(* CODESYS project cl_greenhouseobjectslibrary.library
   Author: Massimo Lucano
   Placeholder: CL_GreenhouseObjects
   Title: CL_GreenhouseObjectsLibrary
   Version: 1.3.3
   Description: library containing all class related to Greenhouse harware objects
   Company: CleanGreensSA

Project tree, tasks and I/O mapping:
  libraries: DefectManager_class, * (CleanGreensSA); Tc2_Standard, * (Beckhoff Automation GmbH); Tc2_System, * (Beckhoff Automation GmbH); Tc3_Module, * (Beckhoff Automation GmbH)
  DUTs/
    data type E_ModeMachine
    data type E_SeqLoader
    data type E_StateMachine
    data type ST_FrqCnvrCtrl_HWQ
    data type ST_StackLight_HWQ
  GVLs/
    global variables C
  POUs/
    ClassesObjectsHW/
      Classes_greeenhouse_20240729/
        function block CL_ButtonBlink [ST]: BlinkOff, BlinkOn, bPressed, Init, LightOff, LightOn
        function block CL_DoubleStopper [ST]: bDesactiveError, bInError, bIsBusyDown, bIsBusyUp, bIsDone, bIsDown, bIsNotDown, bIsUp, Init, InitDefect, ReqDown, ReqUp
        function block CL_Lift_old [ST]: bDesactiveError, bInError, bIsBusyDown, bIsBusyUp, bIsDone, bIsDown, bIsNotDown, bIsUp, Init, ReqDown, ReqUp
        function block CL_LiftStopper [ST]: bDesactiveError, bInError, bIsBusyDown, bIsBusyUp, bIsDone, bIsDown, bIsNotDown, bIsUp, DefectUpdate, Init, InitDefect, ReqDown, ReqUp, Run
        function block CL_LoaderOld [ST]: bInError, bIsBusy, bIsDone, bIsLoad, Init, InitDefect, ReqExtend, ReqLoad, ReqRetract, ReqStop
        function EMPTYSTR2 [ST]
        function FC_TransferPointer [ST]
      function block CL_Ancestor [ST]: Case01Hysto, Case02Hysto, Case03Hysto
      function block CL_Button [ST]: bPressed, Init, LightOff, LightOn
      function block CL_ButtonSafe [ST]: BtnPressed, BtnReleased, Init, LightOff, LightOn
      function block CL_Debug [ST]: Case01Histo, Case02Histo, Case03Histo
      function block CL_FrequencyConverter [ST]: bIsReady, bIsStopped, bSpeedReached, FB_init, Init, ReqMoveBW, ReqMoveFW, ReqReset, ReqStop
      function block CL_GreenhouseSystem [ST]: nModeMachine, nStateMachine, ReqModeMachine
      function block CL_LiftValvesBistableClosed [ST]: bIsBusyDown, bIsBusyUp, bIsDone, bIsDown, bIsUp, Init, ReqDown, ReqUp
      function block CL_SensorFilter [ST]: bStatus, DoNotTouch, FB_init, Init
      function block CL_StackLight [ST]: Init
      function block CL_WaitTimer [ST]: End, Start
      function block CL_WorkbenchRedLight [ST]: BlinkingRed, Init, RedOff, RedOn, Run
      function block CL_WorkbenchSensor [ST]: Init, isModule
      function block CL_WorkbenchStackLight [ST]: Blink, BlinkingOrange, Green, Init, Orange, redOnly, startBlinkingError, stopBlinkingError
  VISUs/
*)

// DUTs/E_ModeMachine
{attribute 'qualified_only'}
{attribute 'strict'}
TYPE E_ModeMachine :
(
  Automatic := 0,
  Manual,
  Startup,
  Setup,
  Maintenance,
  Disabled
);
END_TYPE

// DUTs/E_SeqLoader
{attribute 'qualified_only'}
{attribute 'strict'}
TYPE E_SeqLoader :
(
  cIdle           := 0,
  cStartExtend       ,
  cMovingExtend      ,
  cTargetReached      ,
  cStartRetract      ,
  cMovingRetract     ,
  cEndMovement        ,
  cError
);
END_TYPE

// DUTs/E_StateMachine
{attribute 'qualified_only'}
{attribute 'strict'}
TYPE E_StateMachine :
(
  cIdle := 0,
  cStarting,
  cExecute,
  cStopping,
  cStopped,
  cAborting,
  cAborted,
  cClearing,
  cResetting,
  cInitialization := 255        
);
END_TYPE

// DUTs/ST_FrqCnvrCtrl_HWQ
TYPE ST_FrqCnvrCtrl_HWQ :
STRUCT
  bMoveFW_gq     : BOOL;
  bMoveBW_gq     : BOOL;
  bHighSpeed_gq  : BOOL;
  bReset_gq      : BOOL;
END_STRUCT
END_TYPE

// DUTs/ST_StackLight_HWQ
TYPE ST_StackLight_HWQ :
STRUCT
  bBlue     : BOOL;
  bGreen    : BOOL;
  bOrange   : BOOL;
  bRed      : BOOL;
  bBuzzer   : BOOL;
END_STRUCT
END_TYPE

// GVLs/C
{attribute 'qualified_only'}
VAR_GLOBAL CONSTANT 
	//debug
	uiHistoStep_C								        : INT := 50;
	
	//LiftWorkbench Stacklight
	tLWBBlinkHalfPeriod_C               : TIME :=  T#350MS; // Used for every blinking stacklight
	
	//Lift constant
	//tLift_C													    : TIME := T#3S;

  //Lift error constant
	tLiftDown_C 											  : TIME := T#10S;
	tLiftUp_C  												  : TIME := T#10S;

  //Stopper error constant
	tStopperDown_C 											: TIME := T#5S;
	tStopperUp_C  											: TIME := T#5S;

  //Loader Constant
  tLoaderExtand_C                     : TIME := T#20S;
  tLoaderRetract_C                    : TIME := T#15S;

  //debug
	uiHistoryStep_C										  : INT := 50;
END_VAR

// POUs/ClassesObjectsHW/Classes_greeenhouse_20240729/CL_ButtonBlink
FUNCTION_BLOCK PUBLIC CL_ButtonBlink  EXTENDS R_trig
VAR
	bBtnSens_P 		: POINTER TO BOOL;
	bBtnLight_P 	: POINTER TO BOOL;
	bInit 				: BOOL := FALSE;
	bLight			 	: BOOL := FALSE;
	bBlink				: BOOL := FALSE;
  fbBlink     	: TON := (PT := T#0.5S);
	fbBlink2     	: TON := (PT := T#1.0S);
END_VAR

IF bInit THEN 
	SUPER^(CLK := bBtnSens_P^);
	fbBlink2(in := NOT fbBlink2.Q);
	fbBlink(in :=  fbBlink2.IN);
	
	IF bBlink THEN
		bBtnLight_P^:= fbBlink.Q;
	ELSE
		bBtnLight_P^:= bLight;
	END_IF

END_IF

METHOD PUBLIC BlinkOff
VAR_INPUT
END_VAR
IF bInit THEN 
	bBlink := FALSE;
	bLight := FALSE;
END_IF
END_METHOD

METHOD PUBLIC BlinkOn
VAR_INPUT
END_VAR
IF bInit THEN 
	bBlink := TRUE;
	bLight := FALSE;
END_IF
END_METHOD

PROPERTY PUBLIC bPressed : BOOL
GET
IF bInit THEN
	bPressed := SUPER^.Q;
	{IF defined (debug)}
	bPressed := bBtnSens_P^;
	{END_IF}
ELSE
	bPressed := false;
END_IF
END_GET
END_PROPERTY

METHOD PUBLIC Init : BOOL
VAR_INPUT
	bBtnSensPtrIn_P   : POINTER TO BOOL;
	bBtnLightPtrIn_P  : POINTER TO BOOL;
END_VAR
Init := FALSE;
IF NOT bInit THEN
	Init := bInit := bBtnSensPtrIn_P <> 0 AND bBtnLightPtrIn_P <> 0;
	bBtnSens_P := bBtnSensPtrIn_P;
	bBtnLight_P := bBtnLightPtrIn_P;
	bLight := FALSE;
	bBlink := FALSE;
END_IF
END_METHOD

METHOD PUBLIC LightOff
IF bInit THEN 
	bLight := FALSE;
	bBlink := FALSE; 
END_IF
END_METHOD

METHOD PUBLIC LightOn
IF bInit THEN 
	bLight := TRUE;
	bBlink := FALSE;
END_IF
END_METHOD

END_FUNCTION_BLOCK

// POUs/ClassesObjectsHW/Classes_greeenhouse_20240729/CL_DoubleStopper
(*
ExtractorStopper normally UP
PerpendStopper normally DOWN
controlled together by ExtractorDownPerpendUpStoppersVlv
ExtractorStopperDown and PerpendStopperDown
*)

(*
RFIDStopper normally UP
HandoverStopper normally DOWN
controlled together by RFIDDownHandoverUpStoppersVlv
RFIDStopperDown
*)

FUNCTION_BLOCK CL_DoubleStopper
VAR
//Defect
  objTimeOutStopperUp  : CL_Defect; (*	Not used, so no way to check if the object is working or not	*)
  objTimeOutStopperDown: CL_Defect;

//Error Var
	bErrorUp          : BOOL;
	bErrorDown        : BOOL;
  
//Seq management
	nstpMain          : INT := 0;
  nHistoryStm_AR    : ARRAY[0..C.uiHistoryStep_C] OF INT;
  nLastStm          : INT := -1;

//Index	
  i                 : INT;

//Other var 
  bInit             : BOOL;
  
//FBs
	fbTimerStopperUp     : TON ;
	fbErrorStopperDown   : TON := (PT:= C.tStopperDown_C);
	fbErrorStopperUp     : TON := (PT:= C.tStopperUp_C);
	
//Methods Request
	bRequUp           : BOOL;
	bRequDown         : BOOL;
  
// INTERNAL VAR 		
	_bSensorStp1Down					: BOOL;
  _bSensorStp1Down_P       	: POINTER TO BOOL;
  _bSensorStp2Down_P       	: POINTER TO BOOL;//the secondary stopper could have a down sensor
  _bValveUp_P          			: POINTER TO BOOL;
	
  _objGHSystem_P  : POINTER TO CL_GreenhouseSystem;
  _bIsBusy             : BOOL;
  _bIsBusyUP           : BOOL;
  _bIsBusyDown         : BOOL;
	_bIsDone             : BOOL;
  _bDesactiveError     : BOOL;
  _nLineNumber_P       : POINTER TO INT;
END_VAR

VAR CONSTANT
	nIdle_C             : INT := 0;
	WaitUP_C            : INT := 1;
	nWaitDown_C         : INT := 2;
	nLiftError_C        : INT := 3;
END_VAR

IF NOT bInit THEN
  RETURN;
END_IF

_bSensorStp1Down := _bSensorStp1Down_P^;

fbTimerStopperUp(IN:= NOT _bSensorStp1Down AND _bValveUp_P^);//sensor is false and valve is power on -> trigger timer IN from false to true rising edge

(*IF NOT _bDesactiveError THEN
	IF _objGHSystem_P^.nModeMachine <> E_ModeMachine.Manual THEN// desactive Error in manual mode
		fbErrorStopperUp(IN:= _bSensorStp1Down AND _bValveUp_P^);//stopper should go down -> if after the selected time Q is true --> stopper error remains UP
		fbErrorStopperDown(IN:= NOT _bSensorStp1Down AND NOT _bValveUp_P^);//stopper should go up -> if after the selected time Q is true --> stopper error remains DOWN
	END_IF
	
//	bErrorUp := fbErrorStopperUp.Q;
//	bErrorDown := fbErrorStopperDown.Q;
	objTimeOutStopperUp();
//	objTimeOutStopperUp.SetState(fbErrorStopperUp.Q);
	objTimeOutStopperDown();
//	objTimeOutStopperDown.SetState(fbErrorStopperDown.Q);
	
	IF bErrorUp OR bErrorDown THEN 
		bRequUP := bRequDown := FALSE;//cancel method request
		_bIsDone := FALSE;
		_bIsBusy := FALSE;
		_bIsBusyDown := FALSE;
		_bIsBusyUP := FALSE;
		nstpMain := nLiftError_C;
	END_IF
END_IF*)


CASE nstpMain OF
  // -------------------------------------------------
  nIdle_C:
    IF bRequUp THEN
      bRequUP := FALSE;
      nstpMain := WaitUP_C;
    ELSIF bRequDown THEN
      bRequDown := FALSE;
      nstpMain := nWaitDown_C;
    END_IF
  
  // -------------------------------------------------
  WaitUP_C:
    //lift is going up; no sensor available -> return true when calibration time elapsed
    _bValveUp_P^ := TRUE; //can power on electro-valve
    IF fbTimerStopperUp.Q  THEN
      //if after the calibrated time the sensor is true -> error lift is still down; error detected with the timer
      nstpMain := nIdle_C;
      _bIsDone := TRUE;
      _bIsBusy := FALSE;
      _bIsBusyUp := FALSE;
    END_IF
  
  // -------------------------------------------------
  nWaitDown_C:
    IF _bSensorStp1Down  THEN //lift is down -> sensor is true
      nstpMain := nIdle_C;
      _bIsDone := TRUE;
      _bIsBusy := FALSE;
      _bIsBusyDown := FALSE;
    ELSE
     _bValveUp_P^ := FALSE; //sensor is false -> can power off electro-valve
    END_IF
    
  // -------------------------------------------------
  nLiftError_C:
    //error handling lift error
    IF NOT bErrorUp AND  NOT bErrorDown THEN
      nstpMain := nIdle_C;
    END_IF
END_CASE

  
//Historization of STM
IF nLastStm <> nstpMain THEN
  nLastStm := nstpMain;
  FOR i := C.uiHistoryStep_C TO 1 BY -1 DO
    nHistoryStm_AR[i] := nHistoryStm_AR[i-1];
  END_FOR
  nHistoryStm_AR[0] := nstpMain;
END_IF

PROPERTY bDesactiveError : bool
GET
bDesactiveError := _bDesactiveError;
END_GET
SET
_bDesactiveError := bDesactiveError;
END_SET
END_PROPERTY

PROPERTY bInError : bool
GET
bInError := fbErrorStopperUp.Q OR fbErrorStopperDown.Q;
END_GET
END_PROPERTY

PROPERTY PUBLIC bIsBusyDown : bool
GET
bIsBusyDown := _bIsBusyDown;
END_GET
END_PROPERTY

PROPERTY PUBLIC bIsBusyUp : bool
GET
bIsBusyUp := _bIsBusyUp;
END_GET
END_PROPERTY

PROPERTY PUBLIC bIsDone : bool
GET
bIsDone := _bIsDone;
END_GET
END_PROPERTY

PROPERTY PUBLIC bIsDown : BOOL
GET
bIsDown := _bSensorStp1Down AND NOT _bValveUp_P^;//lift is in down position -> sensor is true and valve is power off  isIN
END_GET
END_PROPERTY

PROPERTY PUBLIC bIsNotDown : BOOL
GET
bIsNotDown := NOT bIsDown;//lift is not in down position -> sensor is true and valve is power off
END_GET
END_PROPERTY

PROPERTY PUBLIC bIsUp : bool
GET
bIsUp := fbTimerStopperUp.Q ;//elapsed time to assert that the stopper is in up position
{IF defined (debug)}
bIsUp := TRUE ;
{END_IF}
END_GET
END_PROPERTY

METHOD Init : BOOL
VAR_INPUT
  //Obj
  GHSystem_P 	: POINTER TO CL_GreenhouseSystem;
  
  //IO
  bSensorStp1Down_P	: POINTER TO BOOL;
  bSensorStp2Down_P	: POINTER TO BOOL;
  bValveStp1Up_P		: POINTER TO BOOL;

  //Var
	tStp1Up						: TIME;
	
	// Location number
	usiNbLocatStopper			: USINT;
END_VAR

// Class ID: 020
//Init Obj
_objGHSystem_P  := GHSystem_P ;

//Init IO
_bSensorStp1Down_P  := bSensorStp1Down_P;
_bSensorStp2Down_P  := bSensorStp2Down_P;//if set to NULL then no secondary sensor available
_bValveUp_P := bValveStp1Up_P;

//Init Var
Init := FALSE;
//Check Init
IF bSensorStp1Down_P <> 0 AND _bValveUp_P <> 0 AND _objGHSystem_P <> 0 THEN
  //Defect
//  ObjTimeOutStopperUp.Register(gvl.objDefectManager,CidCL.sClassID_DoubleStopper_C[usiNbLocatStopper],CidErr.sErrorIDs_DoubleStopper_C[1]);
//  ObjTimeOutStopperDown.Register(gvl.objDefectManager,CidCL.sClassID_DoubleStopper_C[usiNbLocatStopper],CidErr.sErrorIDs_DoubleStopper_C[2]);
  InitDefect(iNumInst := usiNbLocatStopper); // Conversion from short unsigned to signed integer always possible, so OK.
	
  Init := bInit := TRUE;
	fbTimerStopperUp.PT := tStp1Up;	// Maybe to move inside the InitDefect method
END_IF
END_METHOD

METHOD InitDefect : BOOL
VAR_INPUT
	iNumInst	:	INT;
END_VAR
END_METHOD

METHOD PUBLIC ReqDown : BOOL
ReqDown := FALSE;

IF NOT bInError THEN
  ReqDown := TRUE;
  bRequDown := TRUE;
  _bIsBusy := TRUE;
  _bIsBusyDown := TRUE;
END_IF

_bIsDone := FALSE;
END_METHOD

METHOD ReqUp : BOOL
ReqUp := FALSE;

IF NOT bInError THEN
  ReqUp := TRUE;
  bRequUp := TRUE;
  _bIsBusy := TRUE;
  _bIsBusyUp := TRUE;
END_IF

_bIsDone := FALSE;
END_METHOD

END_FUNCTION_BLOCK

// POUs/ClassesObjectsHW/CL_GreenhouseSystem
FUNCTION_BLOCK CL_GreenhouseSystem extends CL_Ancestor
VAR_INPUT
END_VAR
VAR_OUTPUT
END_VAR
VAR
  nLastStateMachine         : E_StateMachine;
  nHistoStateMachine_AR     : ARRAY[0..100]OF E_StateMachine;
  //z                         : UINT;
  
  //INTERNAL VAR
  _nRequestModeMachine      : E_ModeMachine := E_ModeMachine.Automatic;
  _nModeMachine             : E_ModeMachine := E_ModeMachine.Automatic;
  _nStateMachine            : E_StateMachine := E_StateMachine.cIdle;
END_VAR

//State machine histroy
IF nLastStateMachine <> nStateMachine THEN
  nLastStateMachine := nStateMachine;  
  Case01Hysto(nStateMachine);
END_IF

//Manage Mode machine
IF _nRequestModeMachine <> nModeMachine AND _nStateMachine = E_StateMachine.cStopped THEN
	_nModeMachine := _nRequestModeMachine;
END_IF

PROPERTY nModeMachine : E_ModeMachine
GET
nModeMachine := _nModeMachine;
END_GET
SET
_nModeMachine := nModeMachine;
END_SET
END_PROPERTY

PROPERTY nStateMachine : E_StateMachine
GET
nStateMachine := _nStateMachine;
END_GET
SET
_nStateMachine := nStateMachine;
END_SET
END_PROPERTY

METHOD ReqModeMachine : BOOL
VAR_INPUT
  nModeMachine   :E_ModeMachine;
END_VAR
_nRequestModeMachine := nModeMachine;
END_METHOD

END_FUNCTION_BLOCK

// POUs/ClassesObjectsHW/CL_Ancestor
FUNCTION_BLOCK CL_Ancestor
VAR
	i01                         : INT;
  nHistoryStep_AR01           : ARRAY[0..C.uiHistoStep_C] OF DINT;
  nLastStep01                 : DINT := -1;
  
  i02                         : INT;
  nHistoryStep_AR02           : ARRAY[0..C.uiHistoStep_C] OF DINT;
  nLastStep02                 : DINT := -1;
  
  i03                         : INT;
  nHistoryStep_AR03           : ARRAY[0..C.uiHistoStep_C] OF DINT;
  nLastStep03                 : DINT := -1;
END_VAR

METHOD Case01Hysto : BOOL
VAR_INPUT
	nStep : DINT;
END_VAR
IF nStep <> nLastStep01 THEN
  nLastStep01 := nStep;
  FOR i01:= C.uiHistoStep_C TO 1 BY -1 DO
    nHistoryStep_AR01[i01] := nHistoryStep_AR01[i01-1];
  END_FOR
  nHistoryStep_AR01[0] := nStep;
END_IF
END_METHOD

METHOD Case02Hysto : BOOL
VAR_INPUT
	nStep : DINT;
END_VAR
IF nStep <> nLastStep02 THEN
  nLastStep02 := nStep;
  FOR i02:= C.uiHistoStep_C TO 1 BY -1 DO
    nHistoryStep_AR02[i02] := nHistoryStep_AR01[i02-1];
  END_FOR
  nHistoryStep_AR02[0] := nStep;
END_IF
END_METHOD

METHOD Case03Hysto : BOOL
VAR_INPUT
	nStep : DINT;
END_VAR
IF nStep <> nLastStep03 THEN
  nLastStep03 := nStep;
  FOR i03:= C.uiHistoStep_C TO 1 BY -1 DO
    nHistoryStep_AR03[i03] := nHistoryStep_AR01[i03-1];
  END_FOR
  nHistoryStep_AR03[0] := nStep;
END_IF
END_METHOD

END_FUNCTION_BLOCK

// POUs/ClassesObjectsHW/Classes_greeenhouse_20240729/CL_Lift_old
FUNCTION_BLOCK CL_Lift_old
VAR
//Defect
  objTimeOutLiftUp  : CL_Defect;
  objTimeOutLiftDown: CL_Defect;

//Error Var
	bErrorUp          : BOOL;
	bErrorDown        : BOOL;
  
//Seq management
	nstpMain          : INT := 0;
  nHistoryStm_AR    : ARRAY[0..C.uiHistoryStep_C] OF INT;
  nLastStm          : INT := -1;

//Index	
	i                	: UINT;
  hi                : INT;

//Other var 
  bInit             : BOOL;
  
//FBs
	fbTimerLiftUp     : TON ;
	fbErrorLiftDown   : TON := (PT:= C.tLiftDown_C);
	fbErrorLiftUp     : TON := (PT:= C.tLiftUp_C);
	
//Methods Request
	bRequUp           : BOOL;
	bRequDown         : BOOL;
  
// INTERNAL VAR 
  _bSensorDown_P       : POINTER TO BOOL;
  _bValveUp_P          : POINTER TO BOOL;
  _objGHSystem_P  : POINTER TO CL_GreenhouseSystem;
  _bIsBusy             : BOOL;
  _bIsBusyUP           : BOOL;
  _bIsBusyDown         : BOOL;
	_bIsDone             : BOOL;
  _bDesactiveError     : BOOL;
  _nLineNumber_P       : POINTER TO INT;
END_VAR

VAR CONSTANT
	nIdle_C             : INT := 0;
	WaitUP_C            : INT := 1;
	nWaitDown_C         : INT := 2;
	nLiftError_C        : INT := 3;
END_VAR

IF NOT bInit THEN
  RETURN;
END_IF

fbTimerLiftUp(IN:= NOT _bSensorDown_P^ AND _bValveUp_P^);//sensor is false and valve is power on -> trigger timer IN from false to true rising edge

IF NOT _bDesactiveError THEN
	IF _objGHSystem_P^.nModeMachine <> E_ModeMachine.Manual THEN// desactive Error in manual mode
		fbErrorLiftUp(IN:= _bSensorDown_P^ AND _bValveUp_P^);//lift should going down -> if after the selected time Q is true --> lift error remains UP
		fbErrorLiftDown(IN:= NOT _bSensorDown_P^ AND NOT _bValveUp_P^);//lift should going up -> if after the selected time Q is true --> lift error remains DOWN
	END_IF
	
	bErrorUp := fbErrorLiftUp.Q;
	bErrorDown := fbErrorLiftDown.Q;
	ObjTimeOutLiftUp();
	ObjTimeOutLiftUp.Set(fbErrorLiftUp.Q);
	ObjTimeOutLiftDown();
	ObjTimeOutLiftDown.Set(fbErrorLiftDown.Q);
	
	IF bErrorUp OR bErrorDown THEN 
		bRequUP := bRequDown := FALSE;//cancel method request
		_bIsDone := FALSE;
		_bIsBusy := FALSE;
		_bIsBusyDown := FALSE;
		_bIsBusyUP := FALSE;
		nstpMain := nLiftError_C;
	END_IF
end_if


CASE nstpMain OF
  // -------------------------------------------------
  nIdle_C:
    IF bRequUp THEN
      bRequUP := FALSE;
      nstpMain := WaitUP_C;
    ELSIF bRequDown THEN
      bRequDown := FALSE;
      nstpMain := nWaitDown_C;
    END_IF
  
  // -------------------------------------------------
  WaitUP_C:
    //lift is going up; no sensor available -> return true when calibration time elapsed
    _bValveUp_P^ := TRUE; //can power on electro-valve
    IF fbTimerLiftUp.Q  THEN
      //if after the calibrated time the sensor is true -> error lift is still down; error detected with the timer
      nstpMain := nIdle_C;
      _bIsDone := TRUE;
      _bIsBusy := FALSE;
      _bIsBusyUp := FALSE;
    END_IF
  
  // -------------------------------------------------
  nWaitDown_C:
    IF _bSensorDown_P^  THEN //lift is down -> sensor is true
      nstpMain := nIdle_C;
      _bIsDone := TRUE;
      _bIsBusy := FALSE;
      _bIsBusyDown := FALSE;
    ELSE
     _bValveUp_P^ := FALSE; //sensor is false -> can power off electro-valve
    END_IF
    
  // -------------------------------------------------
  nLiftError_C:
    //error handling lift error
    IF NOT bErrorUp AND  NOT bErrorDown THEN
      nstpMain := nIdle_C;
    END_IF
END_CASE

  
//Historization of STM
IF nLastStm <> nstpMain THEN
  nLastStm := nstpMain;
  FOR hi := C.uiHistoryStep_C TO 1 BY -1 DO
    nHistoryStm_AR[hi] := nHistoryStm_AR[hi-1];
  END_FOR
  nHistoryStm_AR[0] := nstpMain;
END_IF

PROPERTY bDesactiveError : bool
GET
bDesactiveError := _bDesactiveError;
END_GET
SET
_bDesactiveError := bDesactiveError;
END_SET
END_PROPERTY

PROPERTY bInError : bool
GET
bInError := fbErrorLiftUp.Q or fbErrorLiftDown.Q;
END_GET
END_PROPERTY

PROPERTY PUBLIC bIsBusyDown : bool
GET
bIsBusyDown := _bIsBusyDown;
END_GET
END_PROPERTY

PROPERTY PUBLIC bIsBusyUp : bool
GET
bIsBusyUp := _bIsBusyUp;
END_GET
END_PROPERTY

PROPERTY PUBLIC bIsDone : bool
GET
bIsDone := _bIsDone;
END_GET
END_PROPERTY

PROPERTY PUBLIC bIsDown : BOOL
GET
bIsDown := _bSensorDown_P^ AND NOT _bValveUp_P^;//lift is in down position -> sensor is true and valve is power off  isIN
END_GET
END_PROPERTY

PROPERTY PUBLIC bIsNotDown : BOOL
GET
bIsNotDown := NOT bIsDown;//lift is not in down position -> sensor is true and valve is power off
END_GET
END_PROPERTY

PROPERTY PUBLIC bIsUp : bool
GET
bIsUp := fbTimerLiftUp.Q ;//elapsed time to assert that the lift is in up position
{IF defined (debug)}
//bIsUp := TRUE ;
{END_IF}
END_GET
END_PROPERTY

METHOD Init : BOOL
VAR_INPUT
  //Obj
  objGHSystem_P : POINTER TO CL_GreenhouseSystem;
  
  //IO
  bSensorDown_P	: POINTER TO BOOL;
  bValveUp_P		: POINTER TO BOOL;
  //Var
	tLiftUp				: TIME;
  nLineNumber_P : POINTER TO INT;
END_VAR
//Init Obj
_objGHSystem_P  := objGHSystem_P;

//Init IO
_bSensorDown_P  := bSensorDown_P;
_bValveUp_P := bValveUp_P;

//Init Var
_nLineNumber_P := nLineNumber_P;

Init := FALSE;
//Check Init
IF _bSensorDown_P <> 0 AND _bValveUp_P <> 0 AND _objGHSystem_P <> 0 AND _nLineNumber_P <> 0 THEN
  //Defect
//  ObjTimeOutLiftUp.Register(gvl.objDefectManager,CidCL.sClassID_Lift_C[(_nLineNumber_P^)+C.usiNbLiftOutSpan_C],CidErr.sErrorIDs_Lift_C[1]);
//  ObjTimeOutLiftDown.Register(gvl.objDefectManager,CidCL.sClassID_Lift_C[(_nLineNumber_P^)+C.usiNbLiftOutSpan_C],CidErr.sErrorIDs_Lift_C[2]);
	
	// No InitDefect, since not intended to be used anymore (replaced by CL_Lift_new (which will be renamed CL_Lift in the end)).
//  ObjTimeOutLiftUp.Register(gvl.objDefectManager,CidCL.sClassID_Lift_C[(_nLineNumber_P^)+C.usiNbLiftOutSpan_C],CidErr.sLiftRiseTimeout);
//  ObjTimeOutLiftDown.Register(gvl.objDefectManager,CidCL.sClassID_Lift_C[(_nLineNumber_P^)+C.usiNbLiftOutSpan_C],CidErr.sLiftFallTimeout);
	// Reimplementation of the Defect, to avoid any overflow with the new error Ids for the Lifts
	ObjTimeOutLiftUp.Register(gvl.objDefectManager,CidCL.sClassID_Lift_C[_nLineNumber_P^],CidErr.sLiftRiseTimeout);
  ObjTimeOutLiftDown.Register(gvl.objDefectManager,CidCL.sClassID_Lift_C[_nLineNumber_P^],CidErr.sLiftFallTimeout);
	
  Init := bInit := TRUE;
	fbTimerLiftUp.PT := tLiftUp;
END_IF
END_METHOD

METHOD PUBLIC ReqDown : BOOL
ReqDown := FALSE;

IF NOT bInError THEN
  ReqDown := TRUE;
  bRequDown := TRUE;
  _bIsBusy := TRUE;
  _bIsBusyDown := TRUE;
END_IF

_bIsDone := FALSE;
END_METHOD

METHOD ReqUp : BOOL
ReqUp := FALSE;

IF NOT bInError THEN
  ReqUp := TRUE;
  bRequUp := TRUE;
  _bIsBusy := TRUE;
  _bIsBusyUp := TRUE;
END_IF

_bIsDone := FALSE;
END_METHOD

END_FUNCTION_BLOCK

// POUs/ClassesObjectsHW/Classes_greeenhouse_20240729/CL_LiftStopper
FUNCTION_BLOCK CL_LiftStopper
VAR
//Error Var
	bErrorUp          : BOOL;
	bErrorDown        : BOOL;
  
//Seq management
	nstpMain          : INT := 0;
  nHistoryStm_AR    : ARRAY[0..C.uiHistoryStep_C] OF INT;
  nLastStm          : INT := -1;

//Index	
	i                	: UINT;
  hi                : INT;

//Other var 
  bInit             : BOOL;
  
//FBs
	fbTimerLiftUp     : TON ;
	fbErrorLiftDown   : TON := (PT:= C.tLiftDown_C);
	fbErrorLiftUp     : TON := (PT:= C.tLiftUp_C);
	
//Methods Request
	bRequUp           : BOOL;
	bRequDown         : BOOL;
  
// INTERNAL VAR 
  _bSensorDown_P       : POINTER TO BOOL;
  _bValveUp_P          : POINTER TO BOOL;
  _objGHSystem_P  : POINTER TO CL_GreenhouseSystem;
  _bIsBusy             : BOOL;
  _bIsBusyUP           : BOOL;
  _bIsBusyDown         : BOOL;
	_bIsDone             : BOOL;
  _bDesactiveError     : BOOL;
  _nLineNumber_P       : POINTER TO INT;
	
	// Defect (common to all type of lift)
	objTimeOutAnyLiftUp  : CL_Defect;	// For every single valve, independent lift
  objTimeOutAnyLiftDown: CL_Defect;
END_VAR

VAR CONSTANT
	nIdle_C             : INT := 0;	// To replace by an enum!
	WaitUP_C            : INT := 1;
	nWaitDown_C         : INT := 2;
	nLiftError_C        : INT := 3;
END_VAR

THIS^.Run();

PROPERTY bDesactiveError : bool
GET
bDesactiveError := _bDesactiveError;
END_GET
SET
_bDesactiveError := bDesactiveError;
END_SET
END_PROPERTY

PROPERTY bInError : bool
GET
bInError := fbErrorLiftUp.Q or fbErrorLiftDown.Q;
END_GET
END_PROPERTY

PROPERTY PUBLIC bIsBusyDown : bool
GET
bIsBusyDown := _bIsBusyDown;
END_GET
END_PROPERTY

PROPERTY PUBLIC bIsBusyUp : bool
GET
bIsBusyUp := _bIsBusyUp;
END_GET
END_PROPERTY

PROPERTY PUBLIC bIsDone : bool
GET
bIsDone := _bIsDone;
END_GET
END_PROPERTY

PROPERTY PUBLIC bIsDown : BOOL
GET
bIsDown := _bSensorDown_P^ AND NOT _bValveUp_P^;//lift is in down position -> sensor is true and valve is power off  isIN
END_GET
END_PROPERTY

PROPERTY PUBLIC bIsNotDown : BOOL
GET
bIsNotDown := NOT bIsDown;//lift is not in down position -> sensor is true and valve is power off
END_GET
END_PROPERTY

PROPERTY PUBLIC bIsUp : bool
GET
bIsUp := fbTimerLiftUp.Q ;//elapsed time to assert that the lift is in up position
{IF defined (debug)}
//bIsUp := TRUE ;
{END_IF}
END_GET
END_PROPERTY

METHOD DefectUpdate : BOOL
END_METHOD

METHOD Init : BOOL
VAR_INPUT
  //Obj
  objGHSystem_P : POINTER TO CL_GreenhouseSystem;
  
  //IO
  bSensorDown_P	: POINTER TO BOOL;
  bValveUp_P		: POINTER TO BOOL;
  //Var
	tLiftUp				: TIME;
  nLineNumber_P : POINTER TO INT;
END_VAR
//Init Obj
_objGHSystem_P  := objGHSystem_P;

//Init IO
_bSensorDown_P  := bSensorDown_P;
_bValveUp_P := bValveUp_P;

//Init Var
_nLineNumber_P := nLineNumber_P;

Init := FALSE;
//Check Init
IF _bSensorDown_P <> 0 AND _bValveUp_P <> 0 AND _objGHSystem_P <> 0 AND _nLineNumber_P <> 0 THEN	// Not rightly written
	fbTimerLiftUp.PT := tLiftUp;	// To move inside the InitDefect ? No, but to replace if the same input in any case! Or keep it for sake of clarity.
  THIS^.InitDefect(iNumInst :=  nLineNumber_P^);	// Init to stabilise
	
	// To decide right now, but level to warning
  Init := bInit := TRUE;
END_IF
END_METHOD

METHOD InitDefect : BOOL
VAR_INPUT
	iNumInst	:	INT;
END_VAR
END_METHOD

METHOD PUBLIC ReqDown : BOOL
ReqDown := FALSE;

IF NOT bInError THEN
  ReqDown := TRUE;
  bRequDown := TRUE;
  _bIsBusy := TRUE;
  _bIsBusyDown := TRUE;
END_IF

_bIsDone := FALSE;
END_METHOD

METHOD ReqUp : BOOL
ReqUp := FALSE;

IF NOT bInError THEN
  ReqUp := TRUE;
  bRequUp := TRUE;
  _bIsBusy := TRUE;
  _bIsBusyUp := TRUE;
END_IF

_bIsDone := FALSE;
END_METHOD

METHOD Run : BOOL
VAR_INPUT
END_VAR
IF NOT bInit THEN
  RETURN;
END_IF

fbTimerLiftUp(IN:= NOT _bSensorDown_P^ AND _bValveUp_P^);//sensor is false and valve is power on -> trigger timer IN from false to true rising edge

IF NOT _bDesactiveError THEN
	IF _objGHSystem_P^.nModeMachine <> E_ModeMachine.Manual THEN// desactive Error in manual mode
		fbErrorLiftUp(IN:= _bSensorDown_P^ AND _bValveUp_P^);//lift should going down -> if after the selected time Q is true --> lift error remains UP
		fbErrorLiftDown(IN:= NOT _bSensorDown_P^ AND NOT _bValveUp_P^);//lift should going up -> if after the selected time Q is true --> lift error remains DOWN
	END_IF
	
	bErrorUp := fbErrorLiftUp.Q;
	bErrorDown := fbErrorLiftDown.Q;
	ObjTimeOutAnyLiftUp();
	ObjTimeOutAnyLiftUp.Set(fbErrorLiftUp.Q);
	ObjTimeOutAnyLiftDown();
	ObjTimeOutAnyLiftDown.Set(fbErrorLiftDown.Q);

	
	IF bErrorUp OR bErrorDown THEN 
		bRequUP := bRequDown := FALSE;//cancel method request
		_bIsDone := FALSE;
		_bIsBusy := FALSE;
		_bIsBusyDown := FALSE;
		_bIsBusyUP := FALSE;
		nstpMain := nLiftError_C;
	END_IF
end_if


CASE nstpMain OF
  // -------------------------------------------------
  nIdle_C:
    IF bRequUp THEN
      bRequUP := FALSE;
      nstpMain := WaitUP_C;
    ELSIF bRequDown THEN
      bRequDown := FALSE;
      nstpMain := nWaitDown_C;
    END_IF
  
  // -------------------------------------------------
  WaitUP_C:
    //lift is going up; no sensor available -> return true when calibration time elapsed
    _bValveUp_P^ := TRUE; //can power on electro-valve
    IF fbTimerLiftUp.Q  THEN
      //if after the calibrated time the sensor is true -> error lift is still down; error detected with the timer
      nstpMain := nIdle_C;
      _bIsDone := TRUE;
      _bIsBusy := FALSE;
      _bIsBusyUp := FALSE;
    END_IF
  
  // -------------------------------------------------
  nWaitDown_C:
    IF _bSensorDown_P^  THEN //lift is down -> sensor is true
      nstpMain := nIdle_C;
      _bIsDone := TRUE;
      _bIsBusy := FALSE;
      _bIsBusyDown := FALSE;
    ELSE
     _bValveUp_P^ := FALSE; //sensor is false -> can power off electro-valve
    END_IF
    
  // -------------------------------------------------
  nLiftError_C:
    //error handling lift error
    IF NOT bErrorUp AND  NOT bErrorDown THEN
      nstpMain := nIdle_C;
    END_IF
END_CASE

  
//Historization of STM
IF nLastStm <> nstpMain THEN
  nLastStm := nstpMain;
  FOR hi := C.uiHistoryStep_C TO 1 BY -1 DO
    nHistoryStm_AR[hi] := nHistoryStm_AR[hi-1];
  END_FOR
  nHistoryStm_AR[0] := nstpMain;
END_IF
END_METHOD

END_FUNCTION_BLOCK

// POUs/ClassesObjectsHW/Classes_greeenhouse_20240729/CL_LoaderOld
FUNCTION_BLOCK CL_LoaderOld
VAR
// Defect
  objTimeOutRetractDefect   :CL_Defect;
  objTimeOutExtandDefect    :CL_Defect;
  
// FBs
  fbTimeOutExtand           : TON :=(PT := c.tLoaderExtand_C);
  fbTimeOutRetract          : TON :=(PT := c.tLoaderRetract_C);
  fbTimeBeforeHighSpeed		  : TON := (PT := T#3S);
  fbTrigAbort               : R_TRIG;
  
// Request  
  bRequestLoad              : BOOL := FALSE;
  boRequestRetract          : BOOL := FALSE;
  boRequestExtend           : BOOL := FALSE;
  boOnlyExtend              : BOOL := FALSE;
  
// Seq management  
  nStep                     : INT := 0;
  nHistoryStep_AR           : ARRAY[0..C.uiHistoryStep_C] OF INT;
  nLastStep                 : INT := -1;
    
// Index  
  i                         : UINT;
	hi												: INT;

// Other var
  bInit                     : BOOL;
  
// INTERNAL VAR
  _bSensorIsExtend_P         : POINTER TO BOOL;
  _bSensorIsRetract_P        : POINTER TO BOOL;
  _bIsBusy                   : BOOL;
  _bIsDone                   : BOOL;  
  _bIsLoad                   : BOOL;
  _nLineNumber               : POINTER TO INT;
  
// INTERNAL OBJECT  
  _objPusher_P               : POINTER TO CL_FrequencyConverter;
  _objGHSystem_P     : POINTER TO CL_GreenhouseSystem;
END_VAR

IF NOT bInit THEN
  RETURN;
END_IF

//Call FBs
fbTimeOutExtand();
fbTimeOutRetract();
fbTimeBeforeHighSpeed(in :=nStep = E_SeqLoader.cMovingExtend);

//Defect
ObjTimeOutRetractDefect();
ObjTimeOutRetractDefect.Set(fbTimeOutRetract.Q);
ObjTimeOutExtandDefect();
ObjTimeOutExtandDefect.Set(fbTimeOutExtand.Q);

fbTrigAbort(CLK := _objGHSystem_P^.nStateMachine = E_StateMachine.cAborting);
IF fbTrigAbort.Q THEN
  nStep           := E_SeqLoader.cError;
  bRequestLoad     := FALSE;
  boRequestRetract := FALSE;
  boRequestExtend  := FALSE;
END_IF
IF _objGHSystem_P^.nStateMachine = E_StateMachine.cStopped THEN
  bRequestLoad     := FALSE;
  boRequestRetract := FALSE;
  boRequestExtend  := FALSE;
END_IF

//--------------------------------------------Sequence-----------------------------------------
CASE nStep OF
  // -------------------------------------------------
  E_SeqLoader.cIdle :
    IF boRequestExtend THEN
      boRequestExtend := FALSE;
      boOnlyExtend    := TRUE;
      nStep          := E_SeqLoader.cStartExtend;
     ELSIF boRequestRetract THEN
      boRequestRetract := FALSE;
      nStep          := E_SeqLoader.cStartRetract; 
     ELSIF bRequestLoad  THEN
      bRequestLoad := FALSE;
      nStep        := E_SeqLoader.cStartExtend;
		END_IF
    
  // -------------------------------------------------
  E_SeqLoader.cStartExtend :
    _objPusher_P^.ReqMoveBW(bHighSpeed:= FALSE);
    IF _bSensorIsExtend_P^  THEN
      nStep := E_SeqLoader.cTargetReached;
    ELSIF _objPusher_P^.bSpeedReached THEN       
      nStep := E_SeqLoader.cMovingExtend;
		END_IF
    
  // -------------------------------------------------
  E_SeqLoader.cMovingExtend :
  IF fbTimeBeforeHighSpeed.Q AND NOT _bSensorIsExtend_P^ THEN
	  _objPusher_P^.ReqMoveBW(bHighSpeed:= TRUE);
  END_IF
    IF fbTimeOutExtand.Q THEN
      nStep := E_SeqLoader.cError;
		END_IF
    IF _bSensorIsExtend_P^ THEN  
      _bIsLoad     := TRUE;
      nStep := E_SeqLoader.cTargetReached;
		END_IF
    
  // -------------------------------------------------
  E_SeqLoader.cTargetReached :
    _objPusher_P^.ReqStop();
    IF  _objPusher_P^.bIsStopped THEN
      IF boOnlyExtend THEN
        nStep := E_SeqLoader.cIdle;
        _bIsBusy     := FALSE;
        boOnlyExtend := FALSE;
      ELSE       
        nStep := E_SeqLoader.cStartRetract;
      END_IF
		END_IF
    
  // -------------------------------------------------
  E_SeqLoader.cStartRetract :
    _objPusher_P^.ReqMoveFW(bHighSpeed:= TRUE);
    IF _bSensorIsRetract_P^  THEN
      nStep := E_SeqLoader.cEndMovement;
    ELSIF _objPusher_P^.bSpeedReached THEN       
      nStep := E_SeqLoader.cMovingRetract;
		END_IF
    
  // -------------------------------------------------
  E_SeqLoader.cMovingRetract :
    IF fbTimeOutRetract.Q THEN
      nStep := E_SeqLoader.cError;
		END_IF
    IF _bSensorIsRetract_P^ THEN       
      nStep := E_SeqLoader.cEndMovement;
		END_IF
    
  // -------------------------------------------------
  E_SeqLoader.cEndMovement :
    _objPusher_P^.ReqStop();
    IF _objPusher_P^.bIsStopped THEN
      _bIsBusy  := FALSE;
      _bIsDone  := TRUE;
      nStep  := E_SeqLoader.cIdle;
		END_IF
    
  // -------------------------------------------------
  E_SeqLoader.cError :
    _bIsBusy  := FALSE;
    bRequestLoad := FALSE;
    _objPusher_P^.ReqStop();
    IF NOT _objPusher_P^.bIsReady AND _objPusher_P^.bIsStopped THEN
      _objPusher_P^.ReqReset();
    ELSE
      nStep  := E_SeqLoader.cIdle;
		END_IF
    
END_CASE


//Historization of the sequence
IF nLastStep <> nStep THEN
  nLastStep := nStep;
  FOR hi := C.uiHistoryStep_C TO 1 BY -1 DO
    nHistoryStep_AR[hi] := nHistoryStep_AR[hi-1];
  END_FOR
  nHistoryStep_AR[0] := nStep;
END_IF

PROPERTY bInError : bool
GET
bInError := nStep = E_SeqLoader.cError;
END_GET
END_PROPERTY

PROPERTY bIsBusy : BOOL
GET
bIsBusy := _bIsBusy;
END_GET
END_PROPERTY

PROPERTY bIsDone : BOOL
GET
bIsDone := _bIsDone;
END_GET
END_PROPERTY

PROPERTY bIsLoad : bool
GET
bIsLoad := _bIsLoad;
END_GET
END_PROPERTY

METHOD Init : BOOL
VAR_INPUT
  //Obj
  objPusher_P           : POINTER TO CL_FrequencyConverter;
  objGreenhouseSystem_P : POINTER TO CL_GreenhouseSystem;
  
  //IO
  bSensorIsExtend_P     : POINTER TO BOOL;
  bSensorIsRetract_P    : POINTER TO BOOL;
 
  //Var
  nLineNumber_P         : POINTER TO INT;
END_VAR

// Class ID: 040
//Init Obj
_objPusher_P := objPusher_P;
_objGHSystem_P := objGreenhouseSystem_P;

//Init IO
_bSensorIsExtend_P := bSensorIsExtend_P;
_bSensorIsRetract_P := bSensorIsRetract_P;

//Init Var
_nLineNumber := nLineNumber_P;

//Check Init
IF _objPusher_P <> 0 AND _bSensorIsExtend_P <> 0 AND _bSensorIsRetract_P <> 0 AND _objGHSystem_P <> 0 AND _nLineNumber <> 0 THEN
  //Defect
//  ObjTimeOutRetractDefect.Register(gvl.objDefectManager,CidCL.sClassID_Loader_C[(nLineNumber_P^)],CidErr.sErrorIDs_Loader_C[1]);
//  ObjTimeOutExtandDefect.Register(gvl.objDefectManager,CidCL.sClassID_Loader_C[(nLineNumber_P^)],CidErr.sErrorIDs_Loader_C[2]);
//  // CAUTION: not possible to indicate the line by this way
//  // => Future fix: use the location Infos in the database (maybe by using another stored procedure)
  InitDefect(iNumInst := nLineNumber_P^);
  bInit := TRUE;
END_IF
END_METHOD

METHOD InitDefect : BOOL
VAR_INPUT
	iNumInst	:	INT;
END_VAR
END_METHOD

METHOD ReqExtend : BOOL
VAR_INPUT
END_VAR
ReqExtend := FALSE;

IF _objPusher_P = 0 THEN
  RETURN;
END_IF

IF _objPusher_P^.bIsReady AND NOT bIsBusy AND NOT _bSensorIsExtend_P^ THEN
  ReqExtend      := TRUE;
  
  _bIsBusy        := TRUE;
  _bIsDone        := FALSE;
  _bIsLoad        := FALSE;
  boRequestExtend := TRUE;
END_IF
END_METHOD

METHOD ReqLoad : BOOL
VAR_INPUT
END_VAR
ReqLoad := FALSE;

IF _objPusher_P = 0 THEN
  RETURN;
END_IF

IF _objPusher_P^.bIsReady AND NOT bIsBusy THEN
  ReqLoad       := TRUE;
  
  _bIsBusy        := TRUE;
  _bIsDone        := FALSE;
  _bIsLoad        := FALSE;
  bRequestLoad := TRUE;
END_IF
END_METHOD

METHOD ReqRetract : BOOL
VAR_INPUT
END_VAR
ReqRetract := FALSE;

IF _objPusher_P = 0 THEN
  RETURN;
END_IF

IF _objPusher_P^.bIsReady AND NOT bIsBusy AND NOT _bSensorIsRetract_P^ THEN
  ReqRetract      := TRUE;
  
  _bIsBusy        := TRUE;
  _bIsDone        := FALSE;
  _bIsLoad        := FALSE;
  boRequestRetract := TRUE;
END_IF
END_METHOD

METHOD ReqStop : BOOL
VAR_INPUT
END_VAR
boRequestExtend := FALSE;
boRequestRetract:= FALSE;
bRequestLoad    := FALSE;
_bIsLoad        := FALSE;
nStep           := E_SeqLoader.cEndMovement;
END_METHOD

END_FUNCTION_BLOCK

// POUs/ClassesObjectsHW/CL_FrequencyConverter
FUNCTION_BLOCK CL_FrequencyConverter EXTENDS CL_Ancestor
VAR
  //Actual OP
  bIsBusyMoveBW                   : BOOL;
  bIsBusyMoveFW                   : BOOL;
                                  
  //Request                       
  bRequestMoveBW                  : BOOL;
  bRequestMoveFW                  : BOOL;
  bRequestStop                    : BOOL;
  bRequestHightSpeed              : BOOL;
  bRequestReset                   : BOOL;
 
  //Step state machine                                                                  
  nStep                          : INT := 0;
  
  //Oter var
  i                               : UINT;
  bInit                           : BOOL;
  
  //FB
  fbClearRetry                    : TON:=(pt:=T#5S); 
  fbAccTime                       : TON;
  fbTimeClearing                  : Ton:= (PT:=T#1S);     
  
// INTERNAL VAR
  _bFrqConvReady_P     : POINTER TO BOOL;
  _bFrqConvRunning_P   : POINTER TO BOOL;
  _stFrqConvOutput_P   : POINTER TO ST_FrqCnvrCtrl_HWQ;
  _bSpeedReached                  : BOOL;

  
END_VAR
VAR CONSTANT
  nIdle_C             :INT := 0;
  nMoveToSetPointFW_C :INT := 1;
  nMoveToSetPointBW_C :INT := 2;
  nStopping_C         :INT := 3;
  nClearing_C         :INT := 4;
  nCleared_C          :INT := 5;
END_VAR

//Check pointer
IF not bInit THEN
  RETURN;
END_IF

//Call FB
fbAccTime(in := nStep=nMoveToSetPointFW_C OR nStep=nMoveToSetPointBW_C);
fbTimeClearing(IN := nStep = nCleared_C );

IF NOT _bFrqConvReady_P^  THEN
  _bSpeedReached := FALSE;
END_IF

CASE nStep OF
  // -------------------------------------------------
  nIdle_C:
    IF bRequestReset THEN
      bRequestReset := FALSE;
      nStep := nClearing_C;
    ELSIF bRequestStop THEN
      bRequestStop := FALSE;
      _bSpeedReached := FALSE;
      nStep := nStopping_C;
    ELSIF bRequestMoveFW THEN
      bRequestMoveFW := FALSE;
      nStep := nMoveToSetPointFW_C;
    ELSIF bRequestMoveBW THEN
      bRequestMoveBW := FALSE;
      nStep := nMoveToSetPointBW_C;
		END_IF
    
  // -------------------------------------------------
  nMoveToSetPointFW_C:   
    _stFrqConvOutput_P^.bMoveFW_gq := TRUE;
    _stFrqConvOutput_P^.bHighSpeed_gq := bRequestHightSpeed;
    IF bRequestStop OR NOT _bFrqConvReady_P^ THEN
      bRequestStop:= FALSE;
      nStep := nStopping_C;
    ELSIF fbAccTime.Q THEN
      _bSpeedReached := TRUE;
      nStep := nIdle_C;
		END_IF  

  // -------------------------------------------------
  nMoveToSetPointBW_C:   
    _stFrqConvOutput_P^.bMoveBW_gq := TRUE;
    _stFrqConvOutput_P^.bHighSpeed_gq := bRequestHightSpeed ;
    IF bRequestStop OR NOT _bFrqConvReady_P^ THEN
      bRequestStop:= FALSE;
      nStep := nStopping_C;
    ELSIF fbAccTime.Q THEN
      _bSpeedReached := TRUE;
      nStep := nIdle_C;
		END_IF 
    
  // -------------------------------------------------
  nStopping_C:
    _stFrqConvOutput_P^.bMoveBW_gq := FALSE;
    _stFrqConvOutput_P^.bMoveFW_gq := FALSE;
    _stFrqConvOutput_P^.bHighSpeed_gq := FALSE;
    IF NOT _bFrqConvRunning_P^ THEN
      nStep := nIdle_C;
      bisBusyMoveBW  := FALSE;
      bIsBusyMoveFW  := FALSE;
    END_IF   
    
  // -------------------------------------------------
  nClearing_C:
    _stFrqConvOutput_P^.bReset_gq := TRUE;
    IF _bFrqConvReady_P^ THEN
      nStep := nCleared_C;
		END_IF  
    
  // -------------------------------------------------
  nCleared_C:
    _stFrqConvOutput_P^.bReset_gq := FALSE;
    IF fbTimeClearing.Q THEN
      nStep := nIdle_C;
    END_IF

END_CASE

Case01Hysto(nStep);

PROPERTY bIsReady : bool
GET
bIsReady := _bFrqConvReady_P^;
END_GET
END_PROPERTY

PROPERTY bIsStopped : bool
GET
bIsStopped := not _bFrqConvRunning_P^;
END_GET
END_PROPERTY

PROPERTY bSpeedReached : bool
GET
bSpeedReached := _bSpeedReached;
END_GET
END_PROPERTY

METHOD FB_init : BOOL
VAR_INPUT
	bInitRetains  : BOOL; // if TRUE, the retain variables are initialized (warm start / cold start)
	bInCopyCode   : BOOL; // if TRUE, the instance afterwards gets moved into the copy code (online change)
  tAccTime      : TIME; // value set inside the frenquency controler
END_VAR
fbAccTime.PT := tAccTime;
END_METHOD

METHOD Init : BOOL
VAR_INPUT
  //IO
  bFrqConvReady_P		: POINTER TO BOOL;
  bFrqConvRunning_P	: POINTER TO BOOL;
  stFrqConv_P				: POINTER TO ST_FrqCnvrCtrl_HWQ;
END_VAR
//Init IO
_bFrqConvReady_P := bFrqConvReady_P;
_bFrqConvRunning_P := bFrqConvRunning_P;
_stFrqConvOutput_P:= stFrqConv_P;

//Check Init
IF _bFrqConvReady_P <> 0 AND _bFrqConvRunning_P <> 0 AND _stFrqConvOutput_P <> 0 THEN
  bInit := TRUE;
END_IF
END_METHOD

METHOD ReqMoveBW : BOOL
VAR_INPUT
  bHighSpeed : BOOL;
END_VAR
ReqMoveBW := FALSE;
IF NOT bIsBusyMoveFW AND _bFrqConvReady_P^ AND (bHighSpeed <> bRequestHightSpeed OR NOT bisBusyMoveBW) THEN
  bisBusyMoveBW        := TRUE;
  ReqMoveBW           := TRUE;
  bRequestMoveBW      := TRUE;
  bRequestHightSpeed  := bHighSpeed;
END_IF
END_METHOD

METHOD ReqMoveFW : BOOL
VAR_INPUT
  bHighSpeed : BOOL;
END_VAR
ReqMoveFW := FALSE;
IF NOT bisBusyMoveBW AND _bFrqConvReady_P^ AND (bHighSpeed <> bRequestHightSpeed OR NOT bisBusyMoveFW) THEN
  ReqMoveFW            := TRUE;
  bRequestMoveFW       := TRUE;
  bisBusyMoveFW        := TRUE;
  bRequestHightSpeed   := bHighSpeed;
END_IF
END_METHOD

METHOD ReqReset : BOOL
VAR_INPUT
END_VAR
ReqReset := FALSE;

IF NOT _bFrqConvReady_P^ AND nStep = nIdle_C THEN
  ReqReset := TRUE;
  bRequestReset := TRUE;
END_IF
END_METHOD

METHOD ReqStop : BOOL
VAR_INPUT
END_VAR
ReqStop := FALSE;
IF nStep <> nStopping_C THEN
  ReqStop := TRUE;
  bRequestStop := TRUE;
END_IF
END_METHOD

END_FUNCTION_BLOCK

// POUs/ClassesObjectsHW/Classes_greeenhouse_20240729/EMPTYSTR2
FUNCTION EMPTYSTR2 : BOOL
VAR_INPUT
	pSTR : POINTER TO STRING;
END_VAR

EMPTYSTR2 := DELETE2(pSTR,pSTR,SIZEOF(pSTR^),LEN2(pSTR),1);

END_FUNCTION

// POUs/ClassesObjectsHW/Classes_greeenhouse_20240729/FC_TransferPointer
//------------------- Custom Automation ----------------------------------------
//******* Nom du programme: FC_PointeurTransfert
//******************************************************************************
//******* Date de création : 23.02.2023           Créateur: Tristan Droz
//*******
//******* Description: Transfert de l'adresse d'un pointeur sur au autre variable tout en la supprimant de la variable précédente
//******************************************************************************

FUNCTION FC_TransferPointer : POINTER TO ST_ModuleData 
VAR_IN_OUT
  stByLocalisation_P : POINTER TO ST_ModuleData;
END_VAR
VAR
END_VAR

FC_TransferPointer := stByLocalisation_P;
stByLocalisation_P := 0;

END_FUNCTION

// POUs/ClassesObjectsHW/CL_Button
FUNCTION_BLOCK PUBLIC CL_Button  EXTENDS R_trig
VAR
	bBtnSens_P : POINTER TO BOOL;
	bBtnLight_P : POINTER TO BOOL;
	bInit : BOOL := FALSE;
	bBtnPressed : BOOL := false;
END_VAR

IF bInit THEN 
	SUPER^(CLK := bBtnSens_P^);
	bBtnLight_P^:= bBtnPressed;
END_IF

PROPERTY PUBLIC bPressed : BOOL
GET
IF bInit THEN
	bPressed := SUPER^.Q;
	{IF defined (simulation)}
	bPressed := bBtnSens_P^;
	{END_IF}
ELSE
	bPressed := false;
END_IF
END_GET
END_PROPERTY

METHOD PUBLIC Init : BOOL
VAR_INPUT
	bBtnSensPtrIn_P   : POINTER TO BOOL;
	bBtnLightPtrIn_P  : POINTER TO BOOL;
END_VAR
Init := FALSE;
IF NOT bInit THEN
	Init := bInit := bBtnSensPtrIn_P <> 0 AND bBtnLightPtrIn_P <> 0;
	bBtnSens_P := bBtnSensPtrIn_P;
	bBtnLight_P := bBtnLightPtrIn_P;
	bBtnPressed := false;
END_IF
END_METHOD

METHOD PUBLIC LightOff
IF bInit THEN 
	bBtnPressed := false;
END_IF
END_METHOD

METHOD PUBLIC LightOn
IF bInit THEN 
	bBtnPressed := TRUE;
END_IF
END_METHOD

END_FUNCTION_BLOCK

// POUs/ClassesObjectsHW/CL_ButtonSafe
FUNCTION_BLOCK PUBLIC CL_ButtonSafe
VAR
	bBtnSens_P  : POINTER TO BOOL;
	bBtnLight_P : POINTER TO BOOL;
	bInit       : BOOL := FALSE;
  bBtnLight   : BOOL;
  
  bBtnRise    : R_trig;
  bBtnFall    : F_trig;
END_VAR

IF bInit THEN 
	bBtnRise(CLK := bBtnSens_P^);
  bBtnFall(CLK := bBtnSens_P^);
  
	bBtnLight_P^:= bBtnLight;
END_IF

PROPERTY PUBLIC BtnPressed : BOOL
GET
IF bInit THEN
	//BtnPressed := bBtnFall.Q;
  BtnPressed := bBtnRise.Q;
	{IF defined (simulation)}
	BtnPressed := bBtnSens_P^;
	{END_IF}
ELSE
	BtnPressed := false;
END_IF
END_GET
END_PROPERTY

PROPERTY PUBLIC BtnReleased : BOOL
GET
IF bInit THEN
	//BtnReleased := bBtnRise.Q;
  BtnReleased := bBtnFall.Q;
	{IF defined (simulation)}
	BtnReleased := bBtnSens_P^;
	{END_IF}
ELSE
	BtnReleased := false;
END_IF
END_GET
END_PROPERTY

METHOD PUBLIC Init : BOOL
VAR_INPUT
	bBtnSensPtrIn_P   : POINTER TO BOOL;
	bBtnLightPtrIn_P  : POINTER TO BOOL;
END_VAR
Init := FALSE;
IF NOT bInit THEN
	Init := bInit := bBtnSensPtrIn_P <> 0 AND bBtnLightPtrIn_P <> 0;
	bBtnSens_P := bBtnSensPtrIn_P;
	bBtnLight_P := bBtnLightPtrIn_P;
	bBtnLight := FALSE;
END_IF
END_METHOD

METHOD PUBLIC LightOff
IF bInit THEN 
	bBtnLight := FALSE;
END_IF
END_METHOD

METHOD PUBLIC LightOn
IF bInit THEN 
	bBtnLight := TRUE;
END_IF
END_METHOD

END_FUNCTION_BLOCK

// POUs/ClassesObjectsHW/CL_Debug
FUNCTION_BLOCK CL_Debug
VAR
	i01                         : INT;
  nHistoryStep_AR01           : ARRAY[0..C.uiHistoStep_C] OF DINT;
  nLastStep01                 : DINT := -1;
  
  i02                         : INT;
  nHistoryStep_AR02           : ARRAY[0..C.uiHistoStep_C] OF DINT;
  nLastStep02                 : DINT := -1;
  
  i03                         : INT;
  nHistoryStep_AR03           : ARRAY[0..C.uiHistoStep_C] OF DINT;
  nLastStep03                 : DINT := -1;
END_VAR

METHOD Case01Histo : BOOL
VAR_INPUT
	nStep : DINT;
END_VAR
IF nStep <> nLastStep01 THEN
  nLastStep01 := nStep;
  FOR i01:= C.uiHistoStep_C TO 1 BY -1 DO
    nHistoryStep_AR01[i01] := nHistoryStep_AR01[i01-1];
  END_FOR
  nHistoryStep_AR01[0] := nStep;
END_IF
END_METHOD

METHOD Case02Histo : BOOL
VAR_INPUT
	nStep : DINT;
END_VAR
IF nStep <> nLastStep02 THEN
  nLastStep02 := nStep;
  FOR i02:= C.uiHistoStep_C TO 1 BY -1 DO
    nHistoryStep_AR02[i02] := nHistoryStep_AR01[i02-1];
  END_FOR
  nHistoryStep_AR02[0] := nStep;
END_IF
END_METHOD

METHOD Case03Histo : BOOL
VAR_INPUT
	nStep : DINT;
END_VAR
IF nStep <> nLastStep03 THEN
  nLastStep03 := nStep;
  FOR i03:= C.uiHistoStep_C TO 1 BY -1 DO
    nHistoryStep_AR03[i03] := nHistoryStep_AR01[i03-1];
  END_FOR
  nHistoryStep_AR03[0] := nStep;
END_IF
END_METHOD

END_FUNCTION_BLOCK

// POUs/ClassesObjectsHW/CL_LiftValvesBistableClosed
FUNCTION_BLOCK CL_LiftValvesBistableClosed  //ValveBistableClosed
VAR
	//Methods Request
	bRequUp        : BOOL;
	bRequDown      : BOOL;
  		
	//Private INTERNAL VAR not accesible
  //IO
  _bValveDown_P : POINTER TO BOOL;
  _bValveUp_P		: POINTER TO BOOL;
	
	_tDown				: TIME;
	_tUp					: TIME;

	_bIsBusy      : BOOL;
  _bIsBusyUP    : BOOL;
  _bIsBusyDown  : BOOL;
	_bIsDone      : BOOL;

	//FBs
	fbTimDown 		: TON ;
	fbTimUp 			: TON ;

	bInit					: BOOL := FALSE;
	nstpMain      : INT := Idle_C;
	tDown: TIME;
	tUp: TIME;
END_VAR

VAR CONSTANT
	Idle_C        : INT := 0;
	WaitUP_C      : INT := 1;
	WaitDown_C    : INT := 2;
END_VAR

//N.B. no sensor available to check that the valve thus the lift is moving -> not possible to implement any kind of errors handling
IF NOT bInit THEN
  RETURN;
END_IF

fbTimUp(IN:= _bValveUp_P^);//sensor is false and valve is power on -> trigger timer IN from false to true rising edge
fbTimDown(IN:= _bValveDown_P^);//sensor is false and valve is power on -> trigger timer IN from false to true rising edge

CASE nstpMain OF
  // -------------------------------------------------
  Idle_C:
    IF bRequUp THEN
      bRequUP := FALSE;
      fbTimUp.PT := _tUp;
      nstpMain := WaitUP_C;
    ELSIF bRequDown THEN
      bRequDown := FALSE;
      fbTimDown.PT := _tDown;
      nstpMain := WaitDown_C;
    END_IF
  
  // -------------------------------------------------
  WaitUP_C:
    //lift is going up; no sensor available -> return true when calibration time elapsed
    _bValveUp_P^ := TRUE; //can power on electro-valve
		_bValveDown_P^ := FALSE;
    IF fbTimUp.Q  THEN
      //after fbTimUp the lift will be up 
      nstpMain := Idle_C;
      _bIsDone := TRUE;
      _bIsBusy := FALSE;
      _bIsBusyUp := FALSE;
    END_IF
  
	// -------------------------------------------------
  WaitDown_C:
    //lift is going down; no sensor available -> return true when calibration time elapsed
    _bValveUp_P^ := FALSE; //can power on electro-valve
		_bValveDown_P^ := TRUE;
    IF fbTimDown.Q  THEN
      //after fbTimDown the lift will be down 
      nstpMain := Idle_C;
      _bIsDone := TRUE;
      _bIsBusy := FALSE;
      _bIsBusyDown := FALSE;
    END_IF

END_CASE

PROPERTY PUBLIC bIsBusyDown : bool
GET
bIsBusyDown := _bIsBusyDown;
END_GET
END_PROPERTY

PROPERTY PUBLIC bIsBusyUp : bool
GET
bIsBusyUp := _bIsBusyUp;
END_GET
END_PROPERTY

PROPERTY PUBLIC bIsDone : bool
GET
bIsDone := _bIsDone;
END_GET
END_PROPERTY

PROPERTY PUBLIC bIsDown : BOOL
GET
bIsDown := fbTimDown.Q ;//elapsed time to assert that the lift is in up position
END_GET
END_PROPERTY

PROPERTY PUBLIC bIsUp : bool
GET
bIsUp := fbTimUp.Q ;//elapsed time to assert that the lift is in up position
END_GET
END_PROPERTY

METHOD Init : BOOL
VAR_INPUT
	bValveDown_P			: POINTER TO BOOL;
  bValveUp_P				: POINTER TO BOOL;
	
	tDown							: TIME;
	tUp							  : TIME;
END_VAR

(*  CONTRACT  
    
    If:
       - the pointers given as inputs are valid (non-null)
       - the times given as inputs are strictly greater than 0.5s
   Then:
      The init method will copy the inputs to the properties of the object,
      set the times for TON Timers, set bInit to 1 and returns true.
      It ensures that!

*)
// Preconditions check
IF bValveDown_P <> 0 AND bValveUp_P <> 0 AND tDown > T#0.5S AND tUp > T#0.5S THEN
  
  //Init IO
  _bValveDown_P  := bValveDown_P;
  _bValveUp_P := bValveUp_P;
  
  _tDown := tDown;  // For future features.
  _tUp := tUp;
  
  fbTimDown.PT := tDown;
	fbTimUp.PT := tUp;
  
  bInit := TRUE;
  Init  := TRUE;
ELSE
  bInit := FALSE;
  Init  := FALSE;
END_IF


////Init IO
//_bValveDown_P  := bValveDown_P;
//_bValveUp_P := bValveUp_P;

//_tDown := tDown;  // For future features.
//_tUp := tUp;

//Init := FALSE;
////Check Init  //MCO to modify, because preconditions to check before doing any modification (risk of null pointer detection or internal state modification)
//IF _bValveDown_P <> 0 AND _bValveUp_P <> 0 AND _tDown > T#0.5S AND _tUp > T#0.5S THEN
//  //Defect
  
//  Init := bInit := TRUE;
//	fbTimDown.PT := tDown;
//	fbTimUp.PT := tUp;
//END_IF
END_METHOD

METHOD PUBLIC ReqDown : BOOL
ReqDown := TRUE;

bRequDown := TRUE;
_bIsBusyDown := TRUE;

bRequUp := FALSE;
_bIsBusyUP := FALSE;

_bIsBusy := TRUE;
_bIsDone := FALSE;
END_METHOD

METHOD ReqUp : BOOL
ReqUp := TRUE;

bRequDown := FALSE;
_bIsBusyDown := FALSE;

bRequUp := TRUE;
_bIsBusyUP := TRUE;

_bIsBusy := TRUE;
_bIsDone := FALSE;
END_METHOD

END_FUNCTION_BLOCK

// POUs/ClassesObjectsHW/CL_SensorFilter
FUNCTION_BLOCK CL_SensorFilter
VAR
//  FBs
  fbFiltre    : tof;
//Other var
  bInit       : bool;
//INTERNAL VAR
  _bSensor_P   : POINTER TO BOOL;
//use to check if sensor is active and then not possiblew to touch manually
	_bDontTouch	: BOOL;
END_VAR

IF not bInit THEN
  RETURN;
END_IF
fbFiltre(IN:= _bSensor_P^);

PROPERTY PRIVATE bStatus : bool
GET
PUBLIC 
VAR
END_VAR
bStatus := fbFiltre.Q;
{IF defined (simulation)}
bStatus := _bSensor_P^;
{END_IF}
END_GET
END_PROPERTY

PROPERTY PUBLIC DoNotTouch : BOOL
GET
DoNotTouch :=_bDontTouch;
END_GET
SET
_bDontTouch := DoNotTouch;
END_SET
END_PROPERTY

METHOD FB_init : BOOL
VAR_INPUT
	bInitRetains  : BOOL; // if TRUE, the retain variables are initialized (warm start / cold start)
	bInCopyCode   : BOOL;  // if TRUE, the instance afterwards gets moved into the copy code (online change)
  tFiltreTime   : TIME;
END_VAR
fbFiltre.PT := tFiltreTime;
END_METHOD

METHOD Init : BOOL
VAR_INPUT
  //IO
  bSensor_P : POINTER TO BOOL;
END_VAR
//Init IO
_bSensor_P := bSensor_P;
_bDontTouch := FALSE;
IF _bSensor_P <> 0 THEN
  bInit := TRUE;
END_IF
END_METHOD

END_FUNCTION_BLOCK

// POUs/ClassesObjectsHW/CL_StackLight
FUNCTION_BLOCK CL_StackLight
VAR_INPUT
END_VAR
VAR_OUTPUT
END_VAR
VAR
//FBs
  fbFlash2    : TON := (PT := T#2S);
  fbFlash     : TON := (PT := T#1S);

//Other var
  bInit       : bool;

// INTERNAL VAR 
 _stStackLight_P    : POINTER TO ST_StackLight_HWQ;
 _objGreenhouseSystem_P : POINTER TO CL_GreenhouseSystem;
END_VAR

IF NOT bInit THEN
  RETURN;
END_IF
//Call FBs
fbFlash2(in := NOT fbFlash2.Q);
fbFlash(in :=  fbFlash2.IN);

_stStackLight_P^.bBlue     := FALSE;
_stStackLight_P^.bBuzzer   := FALSE;
_stStackLight_P^.bGreen    := FALSE;
_stStackLight_P^.bOrange   := FALSE;
_stStackLight_P^.bRed      := FALSE;

CASE _objGreenhouseSystem_P^.nStateMachine OF
  E_StateMachine.cIdle:
    _stStackLight_P^.bGreen := fbFlash.Q;
  
  E_StateMachine.cStarting:
    _stStackLight_P^.bGreen := TRUE;
    _stStackLight_P^.bBuzzer := TRUE;
  
  E_StateMachine.cExecute:
    _stStackLight_P^.bGreen := TRUE;
  
  E_StateMachine.cStopping:
    _stStackLight_P^.bRed := TRUE;
  
  E_StateMachine.cStopped:
    _stStackLight_P^.bRed := TRUE;
  
  E_StateMachine.cAborting:
    _stStackLight_P^.bRed := fbFlash.Q;
  
  E_StateMachine.cAborted:
    _stStackLight_P^.bRed := fbFlash.Q;
  
  E_StateMachine.cClearing:
    _stStackLight_P^.bRed := fbFlash.Q;
  
  E_StateMachine.cResetting:
    _stStackLight_P^.bRed := TRUE;
END_CASE

METHOD Init : BOOL
VAR_INPUT
  //IO
  stStackLight_P : POINTER TO ST_StackLight_HWQ;
  
  //Obj
  objGreenhouseSystem_P : POINTER TO CL_GreenhouseSystem;
END_VAR
//Init IO
_stStackLight_P := stStackLight_P;
_objGreenhouseSystem_P := objGreenhouseSystem_P;

IF _stStackLight_P <> 0 AND _objGreenhouseSystem_P <> 0 THEN
  bInit := TRUE;
END_IF
END_METHOD

END_FUNCTION_BLOCK

// POUs/ClassesObjectsHW/CL_WaitTimer
FUNCTION_BLOCK PUBLIC CL_WaitTimer EXTENDS TON
VAR
	bInit : BOOL := FALSE;
	bEnd  : BOOL := false;
END_VAR

IF bInit THEN 
	SUPER^();
END_IF

PROPERTY PUBLIC End : BOOL
GET
IF bEnd THEN
	bInit := FALSE;
	SUPER^.IN := FALSE;
	SUPER^();
ELSE
	bEnd := SUPER^.Q;
END_IF
End := bEnd;
END_GET
END_PROPERTY

METHOD PUBLIC Start
VAR_INPUT
	tWaitTime : TIME;
END_VAR
bInit := TRUE;
bEnd := FALSE;

IF SUPER^.ET > T#0S THEN
	SUPER^.IN := FALSE;
	SUPER^();
END_IF

SUPER^.PT := tWaitTime;
SUPER^.IN := TRUE;
END_METHOD

END_FUNCTION_BLOCK

// POUs/ClassesObjectsHW/CL_WorkbenchRedLight
FUNCTION_BLOCK CL_WorkbenchRedLight

VAR
  // Init check boolean
  bInit : BOOL  :=  FALSE;

  _bRdLight_P :         POINTER TO BOOL;
  
  // Timer, activation boolean and blinking light ref for blinking
  lightBlinkTimer:    CL_WaitTimer;
  bAllowBlink:        BOOL              :=  FALSE;
END_VAR

(* Retro-compatibility *)
THIS^.Run();

METHOD PUBLIC BlinkingRed : BOOL
VAR_INPUT
END_VAR
IF bInit THEN
  _bRdLight_P^:=1;
  bAllowBlink :=  TRUE;
  lightBlinkTimer.Start(C.tLWBBlinkHalfPeriod_C);
END_IF
END_METHOD

METHOD PUBLIC Init : BOOL
VAR_INPUT // Assignement of the values from the outside
  bRdLight_P :         POINTER TO BOOL;
END_VAR
Init := FALSE;  // Returned value
IF NOT bInit THEN
  
  // Pointers assignement
  _bRdLight_P := bRdLight_P;
  
  // Values assignement
  _bRdLight_P^ := 0;
  
  bInit := TRUE;
  Init := TRUE;
END_IF
END_METHOD

METHOD PUBLIC RedOff : BOOL
VAR_INPUT
END_VAR
IF bInit THEN
  _bRdLight_P^:=0;
  bAllowBlink :=  FALSE;
END_IF
END_METHOD

METHOD PUBLIC RedOn : BOOL
VAR_INPUT
END_VAR
IF bInit THEN
  _bRdLight_P^:=1;
  bAllowBlink :=  FALSE;
END_IF
END_METHOD

METHOD PUBLIC Run : BOOL
VAR_INPUT
END_VAR
IF bInit AND bAllowBlink THEN
  lightBlinkTimer();
  IF lightBlinkTimer.End THEN
    _bRdLight_P^ := NOT _bRdLight_P^;
    lightBlinkTimer.Start(C.tLWBBlinkHalfPeriod_C);
	END_IF
END_IF
END_METHOD

END_FUNCTION_BLOCK

// POUs/ClassesObjectsHW/CL_WorkbenchSensor
FUNCTION_BLOCK CL_WorkbenchSensor
VAR_INPUT
END_VAR
VAR_OUTPUT
END_VAR
VAR
  bInit : BOOL := FALSE;
  _bSensorRaw_P:  POINTER TO BOOL;
  timeFilter: TON;
  risEdgeDetector:  R_TRIG;
END_VAR

METHOD Init : BOOL
VAR_INPUT
  bSensor_P:  POINTER TO BOOL;
END_VAR
IF (bInit = FALSE) AND (bSensor_P <> 0) THEN
  timeFilter.PT := T#100MS;
  _bSensorRaw_P := bSensor_P;
  bInit := TRUE;
END_IF
END_METHOD

METHOD PUBLIC isModule : BOOL
VAR_INPUT
END_VAR

VAR
  filteredSensor: BOOL;
END_VAR
timeFilter(IN:=_bSensorRaw_P^,PT:=T#100MS,Q=>filteredSensor); // True if signal maintained to 1 long enough
risEdgeDetector(CLK:=filteredSensor,Q=>isModule); // True at the exact rise detection
END_METHOD

END_FUNCTION_BLOCK

// POUs/ClassesObjectsHW/CL_WorkbenchStackLight
FUNCTION_BLOCK CL_WorkbenchStackLight
VAR_INPUT
END_VAR
VAR_OUTPUT
END_VAR
VAR
  // Init check boolean
  bInit : BOOL  :=  FALSE;
  // 3 colours
  _bGrLight_P :         POINTER TO BOOL;
  _bOrLight_P :         POINTER TO BOOL;
  _bRdLight_P :         POINTER TO BOOL;
  
  objRedLight:          CL_WorkbenchRedLight;
  
  // Timer, activation boolean and blinking light ref for blinking
  lightBlinkTimer:    CL_WaitTimer;
  bAllowBlink:        BOOL              :=  FALSE;
  bBlinkLight_P:      POINTER TO BOOL;
  
END_VAR

(*  Has to be cyclically called  *)

IF bInit AND bAllowBlink THEN
  THIS^.Blink(bBlinkLight_P);
END_IF

IF bInit = TRUE THEN
  objRedLight.Run();  // Update of the RedLight object.
END_IF

METHOD PRIVATE Blink : BOOL
VAR_INPUT
  bLight_P  : POINTER TO BOOL;
END_VAR

(*  CONTRACT
    
    If the pointer given as input is valid (non null) and correspond to one of 
    the lights (valid adress), then the function toggles the light each time
    the timer ligthBlinkTimer reaches its end, and immediately restarts it.
  *)
IF bLight_P<>0 AND (bLight_P = _bGrLight_P OR bLight_P = _bOrLight_P OR bLight_P = _bRdLight_P) THEN
  // The pointer is valid and refers to one of the lights
  lightBlinkTimer();  // Is this call necessary?
  IF lightBlinkTimer.End THEN
    bLight_P^ := NOT bLight_P^;
    lightBlinkTimer.Start(C.tLWBBlinkHalfPeriod_C);
	END_IF
  Blink := TRUE;
ELSE
  Blink :=  FALSE;
END_IF
END_METHOD

METHOD PUBLIC BlinkingOrange : BOOL
VAR_INPUT
END_VAR
(*  Implicit contract:
    Preconditions: the method init should have been successfully executed previously  *)
IF bInit = TRUE THEN
  _bGrLight_P^ := 0;
  _bOrLight_P^ := 1;
  // _bRdLight_P^ := 0; // Red light directly managed by dedicated object
  
  bAllowBlink   :=  TRUE;
  bBlinkLight_P :=  _bOrLight_P;
  lightBlinkTimer.Start(C.tLWBBlinkHalfPeriod_C);
END_IF
END_METHOD

METHOD PUBLIC Green : BOOL
VAR_INPUT
END_VAR

(*  Implicit contract:
    Preconditions: the method init should have been successfully executed previously  *)
IF bInit = TRUE THEN
  _bGrLight_P^ := 1;
  _bOrLight_P^ := 0;
  //_bRdLight_P^ := 0;  // Red light directly managed by dedicated object
  
  bAllowBlink   :=  FALSE;
END_IF
END_METHOD

METHOD PUBLIC Init : BOOL
VAR_INPUT // Assignement of the values from the outside
  bGrLight_P :         POINTER TO BOOL;
  bOrLight_P :         POINTER TO BOOL;
  bRdLight_P :         POINTER TO BOOL;
END_VAR
Init := FALSE;  // Returned value
IF NOT bInit THEN
  
  // Pointers assignement
  _bGrLight_P := bGrLight_P;
  _bOrLight_P := bOrLight_P;
  _bRdLight_P := bRdLight_P;
  
  // Init of the Red light object
  objRedLight.Init(bRdLight_P :=  _bRdLight_P);
  
  // Values assignement
  THIS^.Green();
  
  bInit := TRUE;
  Init := TRUE;
END_IF
END_METHOD

METHOD PUBLIC Orange : BOOL
VAR_INPUT
END_VAR
(*  Implicit contract:
    Preconditions: the method init should have been successfully executed previously  *)
IF bInit = TRUE THEN
  _bGrLight_P^ := 0;
  _bOrLight_P^ := 1;
  // _bRdLight_P^ := 0; //// Red light directly managed by dedicated object
  
  bAllowBlink   :=  FALSE;
END_IF
END_METHOD

METHOD PUBLIC redOnly : BOOL
VAR_INPUT
END_VAR
IF bInit = TRUE THEN
  _bGrLight_P^ := 0;
  _bOrLight_P^ := 0;
  objRedLight.RedOn();
  
  bAllowBlink   :=  FALSE;
END_IF
END_METHOD

METHOD PUBLIC startBlinkingError : BOOL
VAR_INPUT
END_VAR
IF bInit = TRUE THEN
  objRedLight.BlinkingRed();
  
END_IF
END_METHOD

METHOD PUBLIC stopBlinkingError : BOOL
VAR_INPUT
END_VAR
IF bInit = TRUE THEN
  objRedLight.RedOff();
END_IF
END_METHOD

END_FUNCTION_BLOCK
